Fanuc KAREL source: kt00005.compact.KL

PROGRAM KT00005
%STACKSIZE=65535
%PRIORITY=65535
%NOLOCKGROUP
VAR
I1 : INTEGER
Y2 : ARRAY[2] OF BYTE
OUT : INTEGER
BEGIN
I1=2
Y2[1]=3
OUT=(I1 + Y2[1])
END KT00005
